FUNCTION_BLOCK ABSTRACT FfuBase EXTENDS TExecution IMPLEMENTS IDevice
VAR_INPUT
END_VAR
VAR_OUTPUT
END_VAR
VAR
	{attribute 'OPC.UA.DA' := '0'}
	_name : STRING;
	{attribute 'OPC.UA.DA' := '0'}
	_deviceID : STRING;				
	{attribute 'OPC.UA.DA' := '0'}	
	_family : DeviceFamily;	
	{attribute 'OPC.UA.DA' := '0'}
	_logger : Logger;
	{attribute 'OPC.UA.DA' := '0'}
	_message : StringBuilder;
	{attribute 'OPC.UA.DA' := '0'}
	_ffuConfig : DeviceConfiguration;	
END_VAR

PROPERTY DeviceID : STRING
GET
DeviceID := _deviceID;
END_GET
SET
_deviceID := DeviceID;
END_SET
END_PROPERTY

PROPERTY Family : DeviceFamily
GET
Family := _family;
END_GET
SET
_family := Family;
END_SET
END_PROPERTY

PROPERTY Name : STRING
GET
Name := _name;
END_GET
SET
_name := Name;
END_SET
END_PROPERTY

METHOD PROTECTED ABSTRACT SetSpeed
VAR_INPUT
	Execute : BOOL;
	SpeedPercent : UINT;
END_VAR
END_METHOD

END_FUNCTION_BLOCK

(* stored: Version 1.1.0.1, ProductVersion 3.1.4024.12
   POU FfuBase: Id {6e4bd828-778e-4a35-a17e-2bf286e13d2e}, SpecialFunc None
   Property DeviceID: Id {696f1bf7-03ca-4271-a31c-8a0990d30e8d}
   Get Get: Id {82300cf4-79ca-414f-ae34-0a6d6d6b212a}
   Set Set: Id {781a85b7-7471-4d52-ba7e-d354315609cd}
   Property Family: Id {49791ea6-1576-44ad-b918-d51dc9f94150}
   Get Get: Id {ba867f48-add3-4c87-a3f7-a57fe8c09207}
   Set Set: Id {79c0f197-18f0-4fea-9bde-6b69ca6be42a}
   Property Name: Id {34d792bb-e071-486b-869d-0a847f06020b}
   Get Get: Id {15d91879-d03e-4728-a6d0-5e4d7c18a3a4}
   Set Set: Id {bbd27c2a-2d8b-4506-bbbe-d8f7c5da8a00}
   Method SetSpeed: Id {72ac4b56-ab38-4a0a-89e7-bebe51ee8c4a} *)
